(* CODESYS project FU_sConcat4BIBO.xml

Project tree, tasks and I/O mapping:
  function FU_sConcat4BIBO [ST]
*)

// FU_sConcat4BIBO
//This functions combines 4 strings
//This is the big output version, it has no limits to input or output size
//The wOutSize must be correct otherwise the function can write to unwanted addresses
// |**Version**|**Author**| **Date** |**Changes**
// | 1         | NSN      | 05-02-19 | Creation
// | 2         | NSN      | 14-10-21 | Changed to pointer based
FUNCTION FU_sConcat4BIBO : BOOL
VAR_INPUT
	sOut		:POINTER TO EASCII;		//Output String
	s1			:POINTER TO EASCII;		//Input String1
	s2			:POINTER TO EASCII;		//Input String2
	s3			:POINTER TO EASCII;		//Input String3
	s4			:POINTER TO EASCII;		//Input String4
END_VAR
VAR_INPUT
	wOutSize	:WORD;					//Output String Size
END_VAR

WHILE wOutSize > 0 DO
	wOutSize		:=		wOutSize - 1;
	IF s1^ <> 0 THEN
		sOut^		:=		s1^;
		s1			:=		s1 + 1;
	ELSIF s2^ <> 0 THEN
		sOut^		:=		s2^;
		s2			:=		s2 + 1;
	ELSIF s3^ <> 0 THEN
		sOut^		:=		s3^;
		s3			:=		s3 + 1;
	ELSIF s4^ <> 0 THEN
		sOut^		:=		s4^;
		s4			:=		s4 + 1;
	ELSE
		EXIT;
	END_IF
	sOut			:=		sOut + 1;
END_WHILE
sOut^				:=		EASCII.Null;

END_FUNCTION
